Universal Robots URScript: T001_qwen2.5-coder_32b_baseline_rep1_retry2.urscript

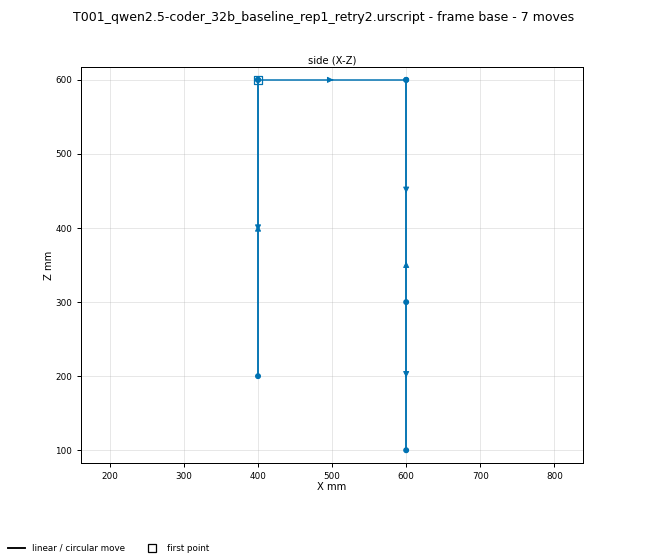
[picture p0: tool path of T001_qwen2.5-coder_32b_baseline_rep1_retry2.urscript in frame base, 7 of 8 moves have a stored position in this frame; points joined in program order, loops and branches not executed]
def simple_pick_place():
    # Set payload parameters
    set_payload(0.5)

    # Move to home position
    movej(get_inverse_kin([0, -1.57, 1.57, -1.57, -1.57, 0]), a=1.2, v=0.3)

    # Approach pick point
    movel(p[0.4, -0.2, 0.6, 3.14, 0, 0], a=1.2, v=0.2)

    # Descend to pick
    movel(p[0.4, -0.2, 0.2, 3.14, 0, 0], a=1.2, v=0.1)

    # Lift from pick
    movel(p[0.4, -0.2, 0.6, 3.14, 0, 0], a=1.2, v=0.15)

    # Transit to place approach
    movel(p[0.6, -0.2, 0.6, 3.14, 0, 0], a=1.2, v=0.2)

    # Approach place point
    movel(p[0.6, -0.2, 0.3, 3.14, 0, 0], a=1.2, v=0.2)

    # Descend to place
    movel(p[0.6, -0.2, 0.1, 3.14, 0, 0], a=1.2, v=0.1)

    # Lift from place
    movel(p[0.6, -0.2, 0.6, 3.14, 0, 0], a=1.2, v=0.15)

end

simple_pick_place()
